FUNCTION "LGF_SplitDWordToWords" : Void
TITLE = LGF_SplitDWordToWords
{ S7_Optimized_Access := 'TRUE' }
AUTHOR : Siemens_Digital_Industry
FAMILY : LGF
NAME : LGF_SplitDWordToWords
//This function splits a DWord variable into 2 Word variables.
   VAR_INPUT
      doubleWord : DWord;   // Bit sequence to be split
   END_VAR

   VAR_OUTPUT
      word1 : Word;   // Output Word 1 - MSW
      word0 : Word;   // Output Word 0 - LSW
   END_VAR


BEGIN
	REGION BLOCK INFO HEADER
	  //===============================================================================
	  // SIEMENS AG / (c)Copyright 2018
	  //-------------------------------------------------------------------------------
	  // Title:            LGF_SplitDWordToWords
	  // Comment/Function: This function splits a DWord variable into 2 Word variables.
	  // Library/Family:   LGF (Library General Functions)
	  // Author:           Siemens Digital Industry Support
	  // Tested with:      S7-PLCSIM Advanced V2.0 SP1
	  // Engineering:      TIA Portal V14 / V14SP1
	  // Restrictions:     ENO disabled - no error handling, no failure possible.
	  // Requirements:     PLC (S7-1200 / S7-1500)
	  //-------------------------------------------------------------------------------
	  // Change log table:
	  // Version  | Date       | Expert in charge       | Changes applied
	  //----------|------------|------------------------|------------------------------
	  // 01.00.00 | 20.06.2019 | Simatic Systems Support
	  //                         First release
	  // 03.00.00 | 23.04.2020 | Simatic Systems Support | Set version to V3.0.0
	  //                         harmonize the version of the whole library
	  // 03.00.01 | 22.02.2021 | Simatic Systems Support
	  //                         Insert documentation
	  //=============================================================================
	END_REGION

	REGION OUTPUT
	  // get the bytes by slice access
	  #word1 := #doubleWord.%W1;
	  #word0 := #doubleWord.%W0;
	  // no error handling needed
	  ENO := TRUE;
	END_REGION

END_FUNCTION

